INTERFACE itfContinuousAxisCommand EXTENDS itfAxisCommand

PROPERTY InVelocity : BOOL
GET
END_GET
END_PROPERTY

END_INTERFACE

(* stored: Version 1.1.0.1, ProductVersion 3.1.4024.11
   Itf itfContinuousAxisCommand: Id {ed80e5f9-1a54-4162-a423-2e4167043dfc}
   Property InVelocity: Id {5e557f79-574b-4480-8944-62a81be74691}
   Get Get: Id {57027170-ebb8-49a0-b747-ff206980d833} *)
